PROGRAM PRG_UpdateRoomTempRh
VAR
END_VAR

(* currently on 0-20mA inputs, but delivering 4-20mA --> need remove 4mA from Signal *)

roomTemp := (INT_TO_REAL(roomTempRaw)/32767.0)*100.0 - 40.0;  (* Sensor Range: -40°C to + 60°C *)
roomRh :=   (INT_TO_REAL(roomRhRaw)/32767.0)*100.0;

END_PROGRAM

(* stored: Version 1.1.0.1, ProductVersion 3.1.4022.7
   POU PRG_UpdateRoomTempRh: Id {eb6dbc51-372c-4e72-b511-be3cc0950038}, SpecialFunc None *)
